{attribute 'GeneratedUsingTerminal: EL9110-0000-0016'}
{attribute addProperty BoxType "EL9110-0000-0016"}
{attribute addProperty Id "InputAT %I*BOOL1"}
{attribute addProperty CRC "2198356929"}
{attribute addProperty Size "1"}
TYPE PowerOK_830843C1 :
STRUCT
	{attribute addProperty Name "Input"}
	Input AT %I* : BOOL;
END_STRUCT
END_TYPE

(* stored: Version 1.2.0.0, ProductVersion 3.1.4024.9
   DUT PowerOK_830843C1: Id {945c1125-6df9-4025-97dd-2043d41882d5} *)
